// Mitsubishi GX Works2 project: Conveyor pause   PLC: FX1N/FX1NC

PROGRAM MAIN
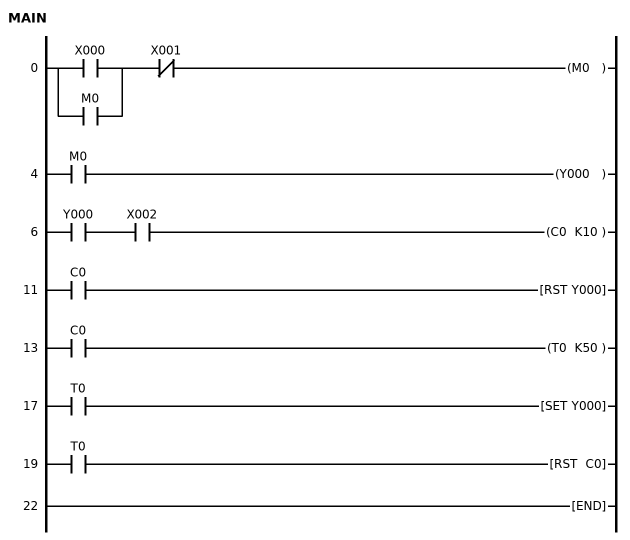
0     LD      X000
      OR      M0
      ANI     X001
      OUT     M0
4     LD      M0
      OUT     Y000
6     LD      Y000
      AND     X002
      OUT     C0 K10
11    LD      C0
      RST     Y000
13    LD      C0
      OUT     T0 K50
17    LD      T0
      SET     Y000
19    LD      T0
      RST     C0
22    END
END_PROGRAM
